FUNCTION_BLOCK ALR_TO_ALR2 (* Composite FB for convert unidirectional ALR to bidirectional ALR2 *)
  (* Standard: 61499-2; Function: ALR_IN publishes its value onto the outgoing (EO1) side of ALR2_BIDIR. Whatever ALR2_BIDIR receives on its incoming (EI1) side is forwarded out again as a plain unidirectional signal via ALR_OUT.; Description: Copyright (c) 2026 HR Agrartechnik GmbH This program and the accompanying materials are made available under the terms of the Eclipse Public License 2.0 which is available at https://www.eclipse.org/legal/epl-2.0/ SPDX-License-Identifier: EPL-2.0 *)
  (* Version 1.0, 2026-09-12, Franz Höpfinger, HR Agrartechnik GmbH, Initial Version - Konvertierungsfamilie vervollstaendigt (analog zu AR2/AB2/AE2). *)
  PACKAGE adapter::conversion::bidirectional;
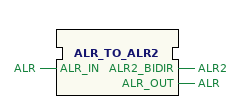
  SOCKETS
    ALR_IN : adapter::types::unidirectional::ALR; (* Adapter Input: unidirectional source *)
  END_SOCKETS
  PLUGS
    ALR2_BIDIR : adapter::types::bidirectional::ALR2; (* Adapter Output: bidirectional tap, outgoing side driven by ALR_IN, incoming side forwarded to ALR_OUT *)
    ALR_OUT : adapter::types::unidirectional::ALR; (* Adapter Output: mirrors ALR2_BIDIR's incoming (request) side *)
  END_PLUGS
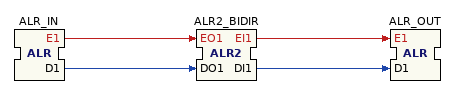
  EVENT_CONNECTIONS
    ALR_IN.E1 TO ALR2_BIDIR.EO1;
    ALR2_BIDIR.EI1 TO ALR_OUT.E1;
  END_CONNECTIONS
  DATA_CONNECTIONS
    ALR_IN.D1 TO ALR2_BIDIR.DO1;
    ALR2_BIDIR.DI1 TO ALR_OUT.D1;
  END_CONNECTIONS
END_FUNCTION_BLOCK
